TYPE ST_System_BSp_Stellwert :
STRUCT
	Anford_Stellventil		: BOOL;
	Anford_Pumpe		: BOOL;
	Anford_Pumpe_Sp	: BOOL;
	Einschaltperiode_Max	: TIME := T#5S;
	Einschalten				: BOOL;
	Modus_Pumpe		: SINT;
	Modus_Pumpe_Sp	: SINT;
	Sollw_Pumpe			: REAL;
	Sollw_Pumpe_Sp		: REAL;
END_STRUCT
END_TYPE

(* stored: Version 1.1.0.1, ProductVersion 3.1.4024.9
   DUT ST_System_BSp_Stellwert: Id {06d1c2a9-3cae-48e0-baef-8f57d3efd910} *)
